FUNCTION_BLOCK CylControlAdp (* Composite Function Block Type *)
  (* Standard: 61499-2 *)
  (* Version 0.0, 7/14/2023, valeriy, nxtControl GmBH, template *)
  PACKAGE Main;
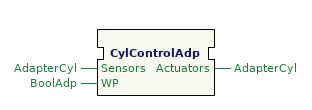
  SOCKETS
    Sensors : AdapterCyl;
    WP : BoolAdp;
  END_SOCKETS
  PLUGS
    Actuators : AdapterCyl;
  END_PLUGS
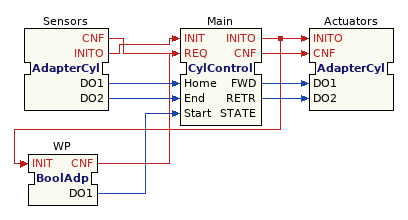
  FBS
    Main : CylControl;
  END_FBS
  EVENT_CONNECTIONS
    Sensors.CNF TO Main.REQ;
    WP.CNF TO Main.REQ;
    Main.INITO TO Actuators.INITO;
    Main.CNF TO Actuators.CNF;
    Sensors.INITO TO Main.INIT;
    Main.INITO TO WP.INIT;
  END_CONNECTIONS
  DATA_CONNECTIONS
    WP.DO1 TO Main.Start;
    Sensors.DO1 TO Main.Home;
    Sensors.DO2 TO Main.End;
    Main.FWD TO Actuators.DO1;
    Main.RETR TO Actuators.DO2;
  END_CONNECTIONS
END_FUNCTION_BLOCK
